TYPE csp_transfer_phase_status_enum :
(		
	CSP_TRANSFER_PHASE_STATUS_START									:= 0,
	CSP_TRANSFER_PHASE_STATUS_DISABLE 								:= 10,
	CSP_TRANSFER_PHASE_STATUS_ENABLE 								:= 20,	
	CSP_TRANSFER_PHASE_STATUS_ENABLED 								:= 30,
	CSP_TRANSFER_PHASE_STATUS_CALCULATE_SLAVE_POSITION_REQUEST		:= 31,
	CSP_TRANSFER_PHASE_STATUS_CALCULATING_SLAVE_POSITION			:= 32,
	CSP_TRANSFER_PHASE_STATUS_REQUEST								:= 33,
	CSP_TRANSFER_PHASE_STATUS_PHASING								:= 34,
	CSP_TRANSFER_PHASE_STATUS_PHASED								:= 35,
	CSP_TRANSFER_PHASE_STATUS_REDEFINE								:= 40,
	CSP_TRANSFER_PHASE_STATUS_REDEFINED								:= 50,
	CSP_TRANSFER_PHASE_STATUS_DONE 									:= 900,
	CSP_TRANSFER_PHASE_STATUS_ERROR 								:= 999
) := CSP_TRANSFER_PHASE_STATUS_START;
END_TYPE

(* stored: Version 1.1.0.1, ProductVersion 3.1.4024.3
   DUT csp_transfer_phase_status_enum: Id {448ceb70-0085-413b-ba7c-c2dd27478aea} *)
